% RSLogix 500 project p2.RSS, saved by version 8.10.00.18 %
PROJECT "P2"    % processor: MicroLogix 1200 %

PROGRAM FILES
  LAD 2 "MAIN"  4 rungs
  LAD 3 "IO 'S"  8 rungs
  LAD 4 "CONTROL"  7 rungs
  LAD 5 "CYCLE'S"  1 rungs

DATA FILES
  O0 OUTPUT  4 elements
  I1 INPUT  4 elements
  S2 STATUS  66 elements
  B3 BINARY  1 elements
  T4 TIMER  1 elements
  C5 COUNTER  1 elements
  R6 CONTROL  1 elements
  N7 INTEGER  1 elements

LADDER 2 "MAIN"
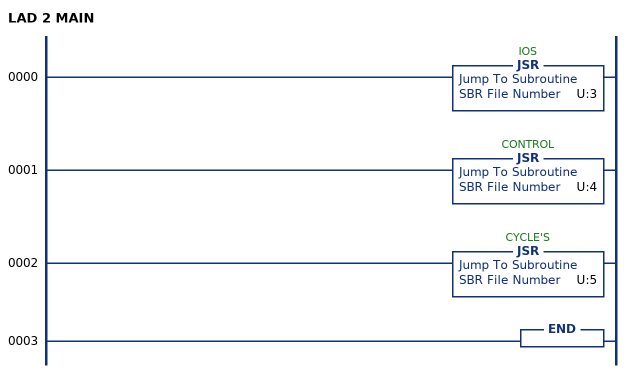
% Rung: 0 %
SOR JSR U:3 EOR
%   U:3  "IOS" %
% Rung: 1 %
SOR JSR U:4 EOR
%   U:4  "CONTROL" %
% Rung: 2 %
SOR JSR U:5 EOR
%   U:5  "CYCLE'S" %
% Rung: 3 %
SOR END EOR

LADDER 3 "IO 'S"
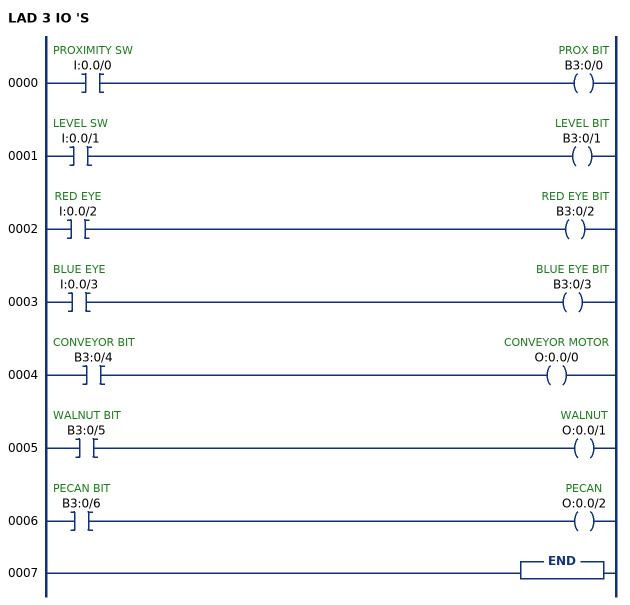
% Rung: 0 %
SOR XIC I:0.0/0 OTE B3:0/0 EOR
%   I:0.0/0  "PROXIMITY SW" %
%   B3:0/0  "PROX BIT" %
% Rung: 1 %
SOR XIC I:0.0/1 OTE B3:0/1 EOR
%   I:0.0/1  "LEVEL SW" %
%   B3:0/1  "LEVEL BIT" %
% Rung: 2 %
SOR XIC I:0.0/2 OTE B3:0/2 EOR
%   I:0.0/2  "RED EYE" %
%   B3:0/2  "RED EYE BIT" %
% Rung: 3 %
SOR XIC I:0.0/3 OTE B3:0/3 EOR
%   I:0.0/3  "BLUE EYE" %
%   B3:0/3  "BLUE EYE BIT" %
% Rung: 4 %
SOR XIC B3:0/4 OTE O:0.0/0 EOR
%   B3:0/4  "CONVEYOR BIT" %
%   O:0.0/0  "CONVEYOR MOTOR" %
% Rung: 5 %
SOR XIC B3:0/5 OTE O:0.0/1 EOR
%   B3:0/5  "WALNUT BIT" %
%   O:0.0/1  "WALNUT" %
% Rung: 6 %
SOR XIC B3:0/6 OTE O:0.0/2 EOR
%   B3:0/6  "PECAN BIT" %
%   O:0.0/2  "PECAN" %
% Rung: 7 %
SOR END EOR

LADDER 4 "CONTROL"
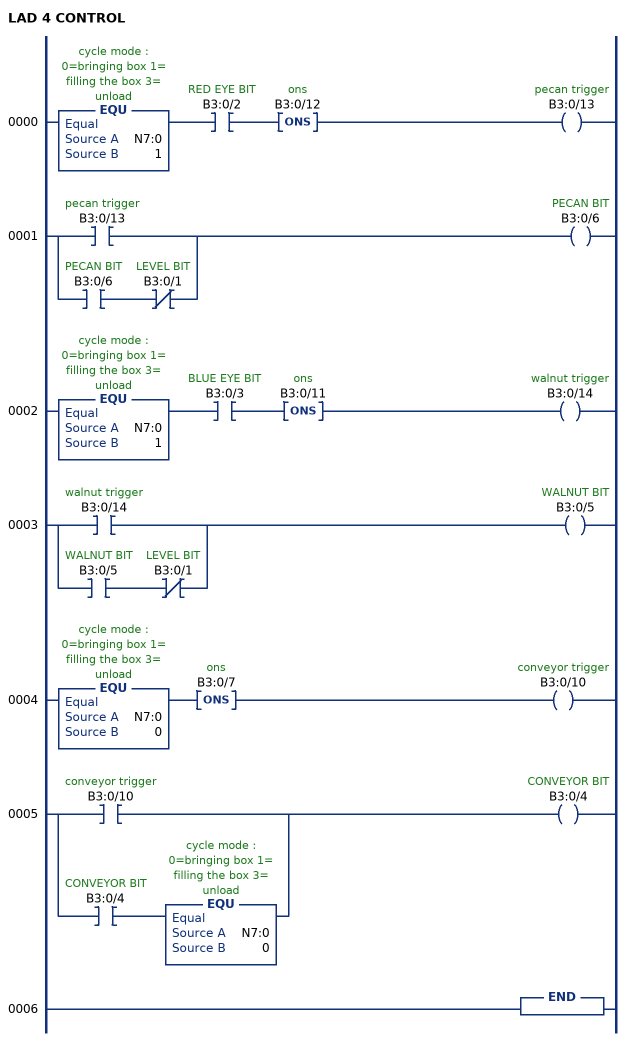
% Rung: 0 %
SOR EQU N7:0 1 XIC B3:0/2 ONS B3:0/12 OTE B3:0/13 EOR
%   N7:0  "cycle mode : 0=bringing box 1= filling the box 3= unload" %
%   B3:0/2  "RED EYE BIT" %
%   B3:0/12  "ons" %
%   B3:0/13  "pecan trigger" %
% Rung: 1 %
SOR BST XIC B3:0/13 NXB XIC B3:0/6 XIO B3:0/1 BND OTE B3:0/6 EOR
%   B3:0/13  "pecan trigger" %
%   B3:0/6  "PECAN BIT" %
%   B3:0/1  "LEVEL BIT" %
% Rung: 2 %
SOR EQU N7:0 1 XIC B3:0/3 ONS B3:0/11 OTE B3:0/14 EOR
%   N7:0  "cycle mode : 0=bringing box 1= filling the box 3= unload" %
%   B3:0/3  "BLUE EYE BIT" %
%   B3:0/11  "ons" %
%   B3:0/14  "walnut trigger" %
% Rung: 3 %
SOR BST XIC B3:0/14 NXB XIC B3:0/5 XIO B3:0/1 BND OTE B3:0/5 EOR
%   B3:0/14  "walnut trigger" %
%   B3:0/5  "WALNUT BIT" %
%   B3:0/1  "LEVEL BIT" %
% Rung: 4 %
SOR EQU N7:0 0 ONS B3:0/7 OTE B3:0/10 EOR
%   N7:0  "cycle mode : 0=bringing box 1= filling the box 3= unload" %
%   B3:0/7  "ons" %
%   B3:0/10  "conveyor trigger" %
% Rung: 5 %
SOR BST XIC B3:0/10 NXB XIC B3:0/4 EQU N7:0 0 BND OTE B3:0/4 EOR
%   B3:0/10  "conveyor trigger" %
%   B3:0/4  "CONVEYOR BIT" %
%   N7:0  "cycle mode : 0=bringing box 1= filling the box 3= unload" %
% Rung: 6 %
SOR END EOR

OTHER DOCUMENTED ADDRESSES
  B3:0/8  "ons 2"
  B3:0/9  "ons 3"

DATA TABLE (non-zero values as saved)
DATA B3
% B3:0 % 0X0090
